// This function has been automatically generated from the project information.
{attribute 'signature_flag' := '1073741824'}
{attribute 'TcGenerated'}
{attribute 'no-analysis'}
FUNCTION F_GetTitle : WSTRING
VAR_INPUT
	
END_VAR

F_GetTitle := "Tc3_Event";

END_FUNCTION

(* stored: Version 1.1.0.1
   POU F_GetTitle: Id {c0f88d1b-0329-4847-a1df-466d1507a1ba}, SpecialFunc None *)
